TYPE MC_ErrorID_Udint : UDINT; END_TYPE

(* stored: Version 1.1.0.1, ProductVersion 3.1.4024.11
   DUT MC_ErrorID_Udint: Id {1b5eb986-6af6-4f73-969d-305461db15b0} *)
